FUNCTION_BLOCK CuttingProcess
VAR_INPUT
	MethodCall : BOOL;
	InputSensor: BOOL;
	CuttingTime : TIME;
	NotAusSignal : BOOL;
	AutomaticMode: BOOL;
END_VAR
VAR_OUTPUT
	CuttingProcess : BOOL;
END_VAR
VAR
//FlipFlop
	RS_CuttingProcess: RS;
//Zeitverzögerung
	TOF_CuttingTime: TOF;
//Flanke	
	R_TRIG_MethodCall: R_TRIG;
END_VAR
VAR // added by the converter: edge detectors and wires of the graphical bodies
    _w1 : BOOL;
END_VAR

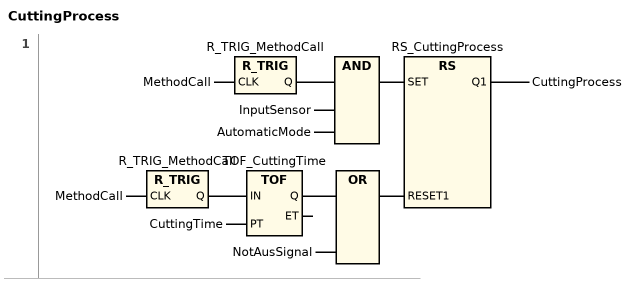
// NETWORK 1
R_TRIG_MethodCall(CLK := MethodCall); // R_TRIG
_w1 := R_TRIG_MethodCall.Q AND InputSensor AND AutomaticMode;
R_TRIG_MethodCall(CLK := MethodCall); // R_TRIG
TOF_CuttingTime(IN := R_TRIG_MethodCall.Q, PT := CuttingTime); // TOF
RS_CuttingProcess(SET := _w1, RESET1 := TOF_CuttingTime.Q OR NotAusSignal); // RS
CuttingProcess := RS_CuttingProcess.Q1;

END_FUNCTION_BLOCK

(* stored: Version 1.1.0.1, ProductVersion 3.1.4024.15
   POU CuttingProcess: Id {21659f6c-d71e-46c8-bac1-8d6b15513317}, SpecialFunc None *)
